// TIA Portal V17 export
// export: Created 2022-02-03T14:45:17.1719495Z, ExportSetting WithDefaults, DisplayName Totally Integrated Automation Portal, DisplayVersion V17, DisplayName TIA Portal Openness, DisplayVersion V17, DisplayName TIA Portal Version Control Interface, DisplayVersion V17, DisplayName SINAMICS Startdrive Advanced, DisplayVersion V17, DisplayName SINAMICS Startdrive G130, G150, S120, S150, SINAMICS MV, S210, DisplayVersion V17, DisplayName SINAMICS Startdrive G110M, G120, G120C, G120D, G120P, G115D, DisplayVersion V17, DisplayName STEP 7 Professional, DisplayVersion V17, DisplayName STEP 7 Safety, DisplayVersion V17, DisplayName WinCC Advanced, DisplayVersion V17
TYPE "typeConveyorOutput"
// stored: Access Published, IsFailsafeCompliant false
   STRUCT
      res0 : Bool;
      P_bay1 : Bool;
      P_bay2 : Bool;
      P_bay3 : Bool;
      P_lightBarrier : Bool;
      K_right : Bool;
      K_left : Bool;
      P_horn : Bool;
   END_STRUCT;
END_TYPE
